FUNCTION_BLOCK FB_ADSHandler
VAR_IN_OUT
	stPalletData			:ST_PalletData;
END_VAR
VAR_INPUT
	sName					:STRING;
	bAck					:BOOL; 				(* Error acknoledge pulse*)
	sAMSNetId				:T_AmsNetID;		(* AMS Net ID *)
	eCommand				:E_ADS_Cmd;			(* ADS command *)
	nIndex					:INT := 1;			(* The index read from the RFID Tag *)
	stEventEntry			:TcEventEntry;		(* Event definition *)	
END_VAR
VAR_OUTPUT
	bBusy					:BOOL;
	bDone					:BOOL;
	bError					:BOOL;
	sError					:STRING(255);		(* Error string *)
	nErrorID				:UDINT;
END_VAR
VAR
	fbReadPalletData		:FB_ReadAdsSymByName;
	fbWritePalletData		:FB_WriteAdsSymByName;
	sPath					:STRING;
	sPathOriginal			:STRING := 'GVL_Persistent.arPaletteData[]'; 
	sEmpty					:STRING:='';
	bIsInitalized			:BOOL;
	fbAlarm					:FB_TcAlarm;
	fbErrorRTrig			:R_Trig;
	fbAckRTrig				:R_Trig;
END_VAR

(*Vezérlés*)
CASE eCommand OF
	NoCmd:		
			fbReadPalletData.bRead := FALSE;
			fbWritePalletData.bWrite := FALSE;
			
	Read:
			fbReadPalletData.bRead := TRUE;
			fbWritePalletData.bWrite := FALSE;
				
	Write:
			fbReadPalletData.bRead := FALSE;
			fbWritePalletData.bWrite := TRUE;				
END_CASE

(*Változónév generálása*)
sPath := INSERT(STR1 := sPathOriginal,
				STR2 := INT_TO_STRING(nIndex),
				POS := FIND(sPathOriginal,'[')
				);

(*ADS kommunikáció*)
fbReadPalletData(
	sNetId:= sAMSNetId, 
	nPort:= 851, 
	sVarName:= sPath , 
	nDestAddr:= ADR(stPalletData), 
	nLen:= SIZEOF(stPalletData));
		
fbWritePalletData( 
	sNetId:= sAMSNetId,
	nPort:= 851, 
	sVarName:= sPath , 
	nSrcAddr:= ADR(stPalletData), 
	nLen:= SIZEOF(stPalletData));

(*Kimenetek beállítása*)
bBusy := fbReadPalletData.bBusy OR fbWritePalletData.bBusy;
bDone :=	(fbReadPalletData.bRead AND NOT fbReadPalletData.bBusy) OR
			(fbWritePalletData.bWrite AND NOT fbWritePalletData.bBusy);

(*Hibaállapotok ellenőrzése*)
IF (fbReadPalletData.bError and fbReadPalletData.bRead) OR (fbWritePalletData.bError and fbWritePalletData.bWrite) THEN
		bError := TRUE;
END_IF
			   
(*Hiba string*)
IF bError THEN
	sError := sName;
	IF		fbReadPalletData.bError THEN
				sError :=  CONCAT(sError, CONCAT('ADS read error. Error code: ',TO_STRING(fbReadPalletData.nErrorId)));
	ELSIF	fbWritePalletData.bError THEN
				sError :=  CONCAT(sError, CONCAT('ADS write error. Error code : ',TO_STRING(fbWritePalletData.nErrorId)));
	END_IF
ELSE
	sError := sEmpty;
END_IF

(*Hiba nyugta*)
IF bAck THEN
	bError := FALSE;
END_IF;

(*Hiba kezelés Tc3_EventLogger*)
IF NOT bIsInitalized THEN
	bIsInitalized := TRUE;
	fbAlarm.CreateEx(stEventEntry, TRUE, 0);
END_IF

fbErrorRTrig(CLK:= bError);
fbAckRTrig(CLK:= bAck);

(*Hiba generálás*)
IF fbErrorRTrig.Q THEN
	fbAlarm.ipArguments.Clear().AddString(sError);
	fbAlarm.Raise(0);
END_IF
(*Hiba nyugtázás*)
IF fbAckRTrig.Q THEN
	fbAlarm.Confirm(0);
END_IF
(*Hiba törlés (nyugtázott és megszűnt)*)
IF fbAlarm.eConfirmationState = 3 AND NOT bError THEN
	fbAlarm.Clear(0, FALSE);
END_IF

END_FUNCTION_BLOCK

(* stored: Version 1.1.0.1, ProductVersion 3.1.4024.10
   POU FB_ADSHandler: Id {6786233a-db71-4d2c-a638-1d74234acd96}, SpecialFunc None *)
